# EPICS substitutions: IOCs/12id/iocBoot/ioc12idd/dac128V.substitutions
file "$(DAC128V)/dac128VApp/Db/singleDAC.db"
{pattern
{P,    D, N, S, PORT,   EGUL,  EGUF, DRVL, DRVH, LOPR, HOPR, PREC,     LINR, VAL}
# Channel 1 is in volts, -10 to 10, with drive limits full range
{12idd:, 1, 1, 0, DAC1,    -10,    10, -10,  10,   -10,  10,   3,    "LINEAR", 0}
# Channel 2 is in volts, -10 to 10, but only allow driving 0 to 10
{12idd:, 1, 2, 1, DAC1,    -10,    10,   -10,  10,     -10,  10,   3,    "LINEAR", 0}
# Channel 3 is in percent of full scale, only allow driving 0 to 100%
{12idd:, 1, 3, 2, DAC1,   -10,   10,   -10, 10,     -10, 10,   3,    "LINEAR", 0}
# Remaing channels are in volts
{12idd:, 1, 4, 3, DAC1,    -10,    10, -10,  10,   -10,  10,   3,    "LINEAR", 0}
{12idd:, 1, 5, 4, DAC1,    -10,    10, -10,  10,   -10,  10,   3,    "LINEAR", 0}
{12idd:, 1, 6, 5, DAC1,    -10,    10, -10,  10,   -10,  10,   3,    "LINEAR", 0}
{12idd:, 1, 7, 6, DAC1,    -10,    10, -10,  10,   -10,  10,   3,    "LINEAR", 0}
{12idd:, 1, 8, 7, DAC1,    -10,    10, -10,  10,   -10,  10,   3,    "LINEAR", 0}

{12idd:, 2, 1, 0, DAC2,    -10,    10, -10,  10,   -10,  10,   3,    "LINEAR", 0}
{12idd:, 2, 2, 1, DAC2,    -10,    10,   -10,  10,     -10,  10,   3,    "LINEAR", 0}
{12idd:, 2, 3, 2, DAC2,   -10,   10,   -10, 10,     -10, 10,   3,    "LINEAR", 0}
{12idd:, 2, 4, 3, DAC2,    -10,    10, -10,  10,   -10,  10,   3,    "LINEAR", 0}
{12idd:, 2, 5, 4, DAC2,    -10,    10, -10,  10,   -10,  10,   3,    "LINEAR", 0}
{12idd:, 2, 6, 5, DAC2,    -10,    10, -10,  10,   -10,  10,   3,    "LINEAR", 0}
{12idd:, 2, 7, 6, DAC2,    -10,    10, -10,  10,   -10,  10,   3,    "LINEAR", 0}
{12idd:, 2, 8, 7, DAC2,    -10,    10, -10,  10,   -10,  10,   3,    "LINEAR", 0}

}
